TYPE U_ExposedLogMsg :
UNION
    sExposedEpicsMessage	: STRING(810);
    arrExposedBuffer 	: ARRAY[0..810] OF BYTE; (* Buffer memory used by FB_MemRingBuffer function block *)
END_UNION
END_TYPE

(* stored: Version 1.1.0.1
   DUT U_ExposedLogMsg: Id {1f914966-33b0-4f8d-ac58-7fae02ae6dc2} *)
